KUKA KRL program: wkz3_ok.src, wkz3_ok.dat

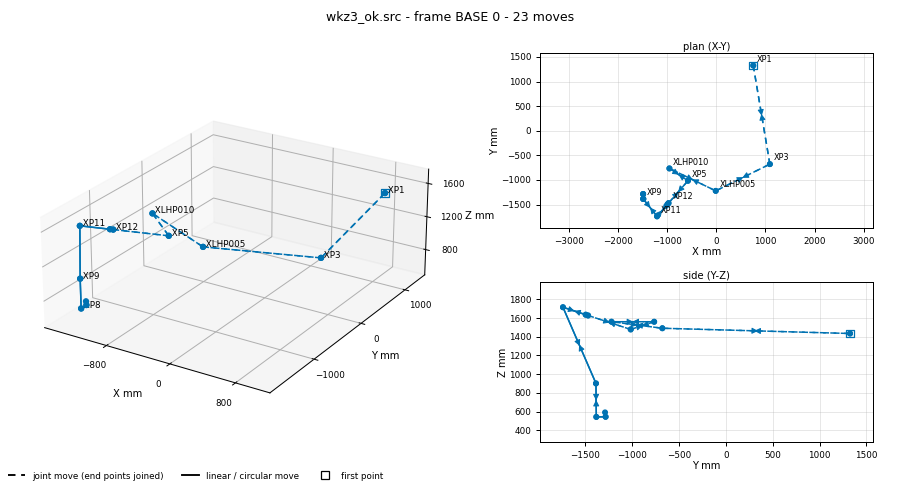
[picture p0: tool path of wkz3_ok.src in frame BASE 0, 23 of 23 moves have a stored position in this frame; points joined in program order, loops and branches not executed]
--- wkz3_ok.src ---
&ACCESS RVP
&REL 455
&COMMENT Check TCP C2
&PARAM DISKPATH = KRC:\R1\Program\TOOL CHANGE
&PARAM TEMPLATE = C:\KRC\Roboter\Template\vorgabe
&PARAM EDITMASK = *
DEF wkz3_ok( )
;FOLD INI
   ;FOLD BASISTECH INI
      GLOBAL INTERRUPT DECL 3 WHEN $STOPMESS==TRUE DO IR_STOPM ( )
      INTERRUPT ON 3
      BAS (#INITMOV,0 )
   ;ENDFOLD (BASISTECH INI)
   ;FOLD SPOTTECH INI
      USERSPOT(#INIT)
   ;ENDFOLD (SPOTTECH INI)
   ;FOLD GRIPPERTECH INI
      USER_GRP(0,DUMMY,DUMMY,GDEFAULT)
   ;ENDFOLD (GRIPPERTECH INI)
   ;FOLD USER INI
      ;Make your modifications here

   ;ENDFOLD (USER INI)
;ENDFOLD (INI)

; Estacao P13.060 - Robo R1
; Programa: Check TCP C2
; Caracterização dos meios de produção:
; 02/09/2014 09:15 Changes by KUKA Roboter do Brasil
;FOLD ; falta instalacao do check vertical;%{PE}%R 8.2.20,%MKUKATPBASIS,%CCOMMENT,%VNORMAL,%P 2:falta  instalacao  do  check  vertical
;ENDFOLD

chk_w3_wechs_ok ( )   ; CHECK FERRAMENTA: GUN C2

;FOLD PTP P1 Vel=100 % PDAT3 Tool[3]:GUN C2 Base[0];%{PE}%R 8.2.20,%MKUKATPBASIS,%CMOVE,%VPTP,%P 1:PTP, 2:P1, 3:, 5:100, 7:PDAT3
$BWDSTART=FALSE
PDAT_ACT=PPDAT3
FDAT_ACT=FP1
BAS(#PTP_PARAMS,100)
PTP XP1
;ENDFOLD
;FOLD PTP P3 Vel=100 % PDAT5 Tool[3]:GUN C2 Base[0];%{PE}%R 8.2.20,%MKUKATPBASIS,%CMOVE,%VPTP,%P 1:PTP, 2:P3, 3:, 5:100, 7:PDAT5
$BWDSTART=FALSE
PDAT_ACT=PPDAT5
FDAT_ACT=FP3
BAS(#PTP_PARAMS,100)
PTP XP3
;ENDFOLD
;FOLD PTP LHP005 CONT Vel=100 % PDAT1 Tool[3]:GUN C2 Base[0];%{PE}%R 8.2.20,%MKUKATPBASIS,%CMOVE,%VPTP,%P 1:PTP, 2:LHP005, 3:C_DIS, 5:100, 7:PDAT1
$BWDSTART=FALSE
PDAT_ACT=PPDAT1
FDAT_ACT=FLHP005
BAS(#PTP_PARAMS,100)
PTP XLHP005 C_DIS
;ENDFOLD
;FOLD PTP LHP010 CONT Vel=100 % PDAT2 Tool[3]:GUN C2 Base[0];%{PE}%R 8.2.20,%MKUKATPBASIS,%CMOVE,%VPTP,%P 1:PTP, 2:LHP010, 3:C_DIS, 5:100, 7:PDAT2
$BWDSTART=FALSE
PDAT_ACT=PPDAT2
FDAT_ACT=FLHP010
BAS(#PTP_PARAMS,100)
PTP XLHP010 C_DIS
;ENDFOLD
;FOLD PTP P5 CONT Vel=100 % PDAT20 Tool[3]:GUN C2 Base[0];%{PE}%R 8.2.20,%MKUKATPBASIS,%CMOVE,%VPTP,%P 1:PTP, 2:P5, 3:C_DIS, 5:100, 7:PDAT20
$BWDSTART=FALSE
PDAT_ACT=PPDAT20
FDAT_ACT=FP5
BAS(#PTP_PARAMS,100)
PTP XP5 C_DIS
;ENDFOLD
;FOLD PTP P12 CONT Vel=100 % PDAT25 Tool[3]:GUN C2 Base[0];%{PE}%R 8.2.20,%MKUKATPBASIS,%CMOVE,%VPTP,%P 1:PTP, 2:P12, 3:C_DIS, 5:100, 7:PDAT25
$BWDSTART=FALSE
PDAT_ACT=PPDAT25
FDAT_ACT=FP12
BAS(#PTP_PARAMS,100)
PTP XP12 C_DIS
;ENDFOLD
;FOLD LIN P13 CONT Vel=0.5 m/s CPDAT13 Tool[3]:GUN C2 Base[0];%{PE}%R 8.2.20,%MKUKATPBASIS,%CMOVE,%VLIN,%P 1:LIN, 2:P13, 3:C_DIS C_DIS, 5:0.5, 7:CPDAT13
$BWDSTART=FALSE
LDAT_ACT=LCPDAT13
FDAT_ACT=FP13
BAS(#CP_PARAMS,0.5)
LIN XP13 C_DIS C_DIS
;ENDFOLD
;FOLD LIN P11 CONT Vel=0.5 m/s CPDAT9 Tool[3]:GUN C2 Base[0];%{PE}%R 8.2.20,%MKUKATPBASIS,%CMOVE,%VLIN,%P 1:LIN, 2:P11, 3:C_DIS C_DIS, 5:0.5, 7:CPDAT9
$BWDSTART=FALSE
LDAT_ACT=LCPDAT9
FDAT_ACT=FP11
BAS(#CP_PARAMS,0.5)
LIN XP11 C_DIS C_DIS
;ENDFOLD
;FOLD LIN P9 CONT Vel=0.5 m/s CPDAT8 Tool[3]:GUN C2 Base[0];%{PE}%R 8.2.20,%MKUKATPBASIS,%CMOVE,%VLIN,%P 1:LIN, 2:P9, 3:C_DIS C_DIS, 5:0.5, 7:CPDAT8
$BWDSTART=FALSE
LDAT_ACT=LCPDAT8
FDAT_ACT=FP9
BAS(#CP_PARAMS,0.5)
LIN XP9 C_DIS C_DIS
;ENDFOLD
;FOLD LIN P8 CONT Vel=0.5 m/s CPDAT10 Tool[3]:GUN C2 Base[0];%{PE}%R 8.2.20,%MKUKATPBASIS,%CMOVE,%VLIN,%P 1:LIN, 2:P8, 3:C_DIS C_DIS, 5:0.5, 7:CPDAT10
$BWDSTART=FALSE
LDAT_ACT=LCPDAT10
FDAT_ACT=FP8
BAS(#CP_PARAMS,0.5)
LIN XP8 C_DIS C_DIS
;ENDFOLD
;FOLD LIN LHP015 Vel=0.5 m/s CPDAT3 Tool[3]:GUN C2 Base[0];%{PE}%R 8.2.20,%MKUKATPBASIS,%CMOVE,%VLIN,%P 1:LIN, 2:LHP015, 3:, 5:0.5, 7:CPDAT3
$BWDSTART=FALSE
LDAT_ACT=LCPDAT3
FDAT_ACT=FLHP015
BAS(#CP_PARAMS,0.5)
LIN XLHP015
;ENDFOLD

;FOLD ; posicao check tcp;%{PE}%R 4.1.16,%MKUKATPBASIS,%CCOMMENT,%VNORMAL,%P 2:posicao check tcp
;ENDFOLD
;FOLD LIN ChkTCPPos_Gun02 Vel=0.5 m/s CPDAT1 Tool[3]:GUN C2 Base[0];%{PE}%R 8.2.20,%MKUKATPBASIS,%CMOVE,%VLIN,%P 1:LIN, 2:ChkTCPPos_Gun02, 3:, 5:0.5, 7:CPDAT1
$BWDSTART=FALSE
LDAT_ACT=LCPDAT1
FDAT_ACT=FChkTCPPos_Gun02
BAS(#CP_PARAMS,0.5)
LIN XChkTCPPos_Gun02
;ENDFOLD
;FOLD WAIT Time= 5 sec;%{PE}%R 4.1.16,%MKUKATPBASIS,%CWAIT,%VWAIT,%P 2:5
WAIT SEC 5
;ENDFOLD

;FOLD LIN P7 CONT Vel=0.5 m/s CPDAT4 Tool[3]:GUN C2 Base[0];%{PE}%R 8.2.20,%MKUKATPBASIS,%CMOVE,%VLIN,%P 1:LIN, 2:P7, 3:C_DIS C_DIS, 5:0.5, 7:CPDAT4
$BWDSTART=FALSE
LDAT_ACT=LCPDAT4
FDAT_ACT=FP7
BAS(#CP_PARAMS,0.5)
LIN XP7 C_DIS C_DIS
;ENDFOLD
;FOLD LIN P14 CONT Vel=0.5 m/s CPDAT11 Tool[3]:GUN C2 Base[0];%{PE}%R 8.2.20,%MKUKATPBASIS,%CMOVE,%VLIN,%P 1:LIN, 2:P14, 3:C_DIS C_DIS, 5:0.5, 7:CPDAT11
$BWDSTART=FALSE
LDAT_ACT=LCPDAT11
FDAT_ACT=FP14
BAS(#CP_PARAMS,0.5)
LIN XP14 C_DIS C_DIS
;ENDFOLD
;FOLD LIN P15 CONT Vel=0.5 m/s CPDAT12 Tool[3]:GUN C2 Base[0];%{PE}%R 8.2.20,%MKUKATPBASIS,%CMOVE,%VLIN,%P 1:LIN, 2:P15, 3:C_DIS C_DIS, 5:0.5, 7:CPDAT12
$BWDSTART=FALSE
LDAT_ACT=LCPDAT12
FDAT_ACT=FP15
BAS(#CP_PARAMS,0.5)
LIN XP15 C_DIS C_DIS
;ENDFOLD
;FOLD LIN P16 CONT Vel=0.5 m/s CPDAT14 Tool[3]:GUN C2 Base[0];%{PE}%R 8.2.20,%MKUKATPBASIS,%CMOVE,%VLIN,%P 1:LIN, 2:P16, 3:C_DIS C_DIS, 5:0.5, 7:CPDAT14
$BWDSTART=FALSE
LDAT_ACT=LCPDAT14
FDAT_ACT=FP16
BAS(#CP_PARAMS,0.5)
LIN XP16 C_DIS C_DIS
;ENDFOLD
;FOLD LIN P17 CONT Vel=0.5 m/s CPDAT15 Tool[3]:GUN C2 Base[0];%{PE}%R 8.2.20,%MKUKATPBASIS,%CMOVE,%VLIN,%P 1:LIN, 2:P17, 3:C_DIS C_DIS, 5:0.5, 7:CPDAT15
$BWDSTART=FALSE
LDAT_ACT=LCPDAT15
FDAT_ACT=FP17
BAS(#CP_PARAMS,0.5)
LIN XP17 C_DIS C_DIS
;ENDFOLD
;FOLD LIN P18 CONT Vel=0.5 m/s CPDAT17 Tool[3]:GUN C2 Base[0];%{PE}%R 8.2.20,%MKUKATPBASIS,%CMOVE,%VLIN,%P 1:LIN, 2:P18, 3:C_DIS C_DIS, 5:0.5, 7:CPDAT17
$BWDSTART=FALSE
LDAT_ACT=LCPDAT17
FDAT_ACT=FP18
BAS(#CP_PARAMS,0.5)
LIN XP18 C_DIS C_DIS
;ENDFOLD
;FOLD PTP P19 CONT Vel=100 % PDAT27 Tool[3]:GUN C2 Base[0];%{PE}%R 8.2.20,%MKUKATPBASIS,%CMOVE,%VPTP,%P 1:PTP, 2:P19, 3:C_DIS, 5:100, 7:PDAT27
$BWDSTART=FALSE
PDAT_ACT=PPDAT27
FDAT_ACT=FP19
BAS(#PTP_PARAMS,100)
PTP XP19 C_DIS
;ENDFOLD
;FOLD PTP P20 CONT Vel=100 % PDAT28 Tool[3]:GUN C2 Base[0];%{PE}%R 8.2.20,%MKUKATPBASIS,%CMOVE,%VPTP,%P 1:PTP, 2:P20, 3:C_DIS, 5:100, 7:PDAT28
$BWDSTART=FALSE
PDAT_ACT=PPDAT28
FDAT_ACT=FP20
BAS(#PTP_PARAMS,100)
PTP XP20 C_DIS
;ENDFOLD
;FOLD PTP P21 CONT Vel=100 % PDAT29 Tool[3]:GUN C2 Base[0];%{PE}%R 8.2.20,%MKUKATPBASIS,%CMOVE,%VPTP,%P 1:PTP, 2:P21, 3:C_DIS, 5:100, 7:PDAT29
$BWDSTART=FALSE
PDAT_ACT=PPDAT29
FDAT_ACT=FP21
BAS(#PTP_PARAMS,100)
PTP XP21 C_DIS
;ENDFOLD
;FOLD PTP P22 CONT Vel=100 % PDAT30 Tool[3]:GUN C2 Base[0];%{PE}%R 8.2.20,%MKUKATPBASIS,%CMOVE,%VPTP,%P 1:PTP, 2:P22, 3:C_DIS, 5:100, 7:PDAT30
$BWDSTART=FALSE
PDAT_ACT=PPDAT30
FDAT_ACT=FP22
BAS(#PTP_PARAMS,100)
PTP XP22 C_DIS
;ENDFOLD
;FOLD PTP P23 CONT Vel=100 % PDAT31 Tool[3]:GUN C2 Base[0];%{PE}%R 8.2.20,%MKUKATPBASIS,%CMOVE,%VPTP,%P 1:PTP, 2:P23, 3:C_DIS, 5:100, 7:PDAT31
$BWDSTART=FALSE
PDAT_ACT=PPDAT31
FDAT_ACT=FP23
BAS(#PTP_PARAMS,100)
PTP XP23 C_DIS
;ENDFOLD
END

--- wkz3_ok.dat ---
&ACCESS RVP
&REL 455
&COMMENT Check TCP C2
&PARAM DISKPATH = KRC:\R1\Program\TOOL CHANGE
&PARAM TEMPLATE = C:\KRC\Roboter\Template\vorgabe
&PARAM EDITMASK = *
DEFDAT  wkz3_ok
;FOLD EXTERNAL DECLARATIONS;%{PE}%MKUKATPBASIS,%CEXT,%VCOMMON,%P
;FOLD GRIPPERTECH EXT
EXT  H50 (INT  :IN,INT  :IN,INT  :IN,GRP_TYP  :IN )
;ENDFOLD (GRIPPERTECH EXT)
;FOLD SPOTTECH EXT
EXT  USERSPOT (S_COMMAND  :IN,SPOT_TYPE  :IN )
;ENDFOLD (SPOTTECH EXT)
;FOLD BASISTECH EXT;%{PE}%MKUKATPBASIS,%CEXT,%VEXT,%P
EXT  BAS (BAS_COMMAND  :IN,REAL  :IN )
DECL INT SUCCESS
;ENDFOLD (BASISTECH EXT)
;FOLD USER EXT;%{E}%MKUKATPUSER,%CEXT,%VEXT,%P
;Make your modifications here

;ENDFOLD (USER EXT)
;ENDFOLD (EXTERNAL DECLARATIONS)

DECL PDAT PPDAT1={VEL 100.0,ACC 80.0,APO_DIST 10.0,APO_MODE #CDIS}
DECL E6POS XLHP010={X -951.651184,Y -765.088989,Z 1560.073,A -119.308197,B -41.8342018,C -84.1509628,S 18,T 2,E1 0.0,E2 0.0,E3 0.0,E4 0.0,E5 0.0,E6 0.0}
DECL FDAT FLHP010={TOOL_NO 3,BASE_NO 0,IPO_FRAME #BASE,TQ_STATE FALSE}
DECL PDAT PPDAT2={VEL 100.0,ACC 80.0,APO_DIST 10.0,APO_MODE #CDIS}
DECL E6POS XLHP015={X -1485.69995,Y -1283.427,Z 545.450623,A 90.8472366,B -0.687042773,C 0.235894397,S 18,T 10,E1 0.0,E2 0.0,E3 0.0,E4 0.0,E5 0.0,E6 0.0}
DECL FDAT FLHP015={TOOL_NO 3,BASE_NO 0,IPO_FRAME #BASE,TQ_STATE FALSE}
DECL E6POS XLHP020={X -1484.229,Y -1382.71899,Z 544.335388,A 90.8472672,B -0.689551473,C 0.235781297,S 18,T 10,E1 0.0,E2 0.0,E3 0.0,E4 0.0,E5 0.0,E6 0.0}
DECL FDAT FLHP020={TOOL_NO 3,BASE_NO 0,IPO_FRAME #BASE,TQ_STATE FALSE}
DECL E6POS XLHP025={X 1034.203,Y -165.537598,Z 959.119873,A -100.153702,B -15.1243601,C -86.5133896,S 18,T 2,E1 0.0,E2 0.0,E3 0.0,E4 0.0,E5 0.0,E6 0.0}
DECL FDAT FLHP025={TOOL_NO 3,BASE_NO 0,IPO_FRAME #BASE,TQ_STATE FALSE}
DECL PDAT PPDAT7={VEL 100.0,ACC 80.0,APO_DIST 10.0,APO_MODE #CDIS}
DECL E6POS XLHP030={X 1218.96802,Y 806.147278,Z 1597.64697,A 176.970596,B -2.82581401,C -90.4064636,S 18,T 3,E1 0.0,E2 0.0,E3 0.0,E4 0.0,E5 0.0,E6 0.0}
DECL FDAT FLHP030={TOOL_NO 3,BASE_NO 0,IPO_FRAME #BASE,TQ_STATE FALSE}
DECL PDAT PPDAT8={VEL 100.0,ACC 80.0,APO_DIST 10.0,APO_MODE #CDIS}
DECL PDAT PPDAT14={VEL 30.0,ACC 80.0,APO_DIST 10.0}
DECL PDAT PPDAT10={VEL 100.0,ACC 80.0,APO_DIST 10.0}
DECL PDAT PPDAT11={VEL 100.0,ACC 80.0,APO_DIST 10.0}
DECL E6POS XLHP005={X -10.4802904,Y -1220.74597,Z 1560.54199,A -68.6302338,B -41.8773613,C -84.0859604,S 18,T 2,E1 0.0,E2 0.0,E3 0.0,E4 0.0,E5 0.0,E6 0.0}
DECL FDAT FLHP005={TOOL_NO 3,BASE_NO 0,IPO_FRAME #BASE,TQ_STATE FALSE}
DECL E6POS XChkTCPPos_Gun02={X -1485.28503,Y -1289.51794,Z 592.772583,A 90.8463516,B -0.690602124,C 0.233830601,S 18,T 34,E1 0.0,E2 0.0,E3 0.0,E4 0.0,E5 0.0,E6 0.0}
DECL FDAT FChkTCPPos_Gun02={TOOL_NO 3,BASE_NO 0,IPO_FRAME #BASE,TQ_STATE FALSE}
DECL BASIS_SUGG_T LAST_BASIS={POINT1[] "P23                     ",POINT2[] "P23                     ",CP_PARAMS[] "CPDAT15                 ",PTP_PARAMS[] "PDAT31                  ",CONT[] "C_DIS                   ",CP_VEL[] "0.5                     ",PTP_VEL[] "100                     ",SYNC_PARAMS[] "SYNCDAT                 ",SPL_NAME[] "S0                      "}
DECL E6POS XP1={X 752.183289,Y 1325.57202,Z 1434.74805,A 80.377739,B -52.962841,C -87.0940628,S 18,T 3,E1 0.0,E2 0.0,E3 0.0,E4 0.0,E5 0.0,E6 0.0}
DECL FDAT FP1={TOOL_NO 3,BASE_NO 0,IPO_FRAME #BASE,POINT2[] " ",TQ_STATE FALSE}
DECL PDAT PPDAT3={VEL 100.0,ACC 100.0,APO_DIST 100.0,APO_MODE #CDIS,GEAR_JERK 50.0}
DECL E6POS XP2={X 752.183411,Y 1325.57202,Z 1434.74805,A 80.3777237,B -52.9628296,C -87.0940475,S 18,T 3,E1 0.0,E2 0.0,E3 0.0,E4 0.0,E5 0.0,E6 0.0}
DECL FDAT FP2={TOOL_NO 3,BASE_NO 0,IPO_FRAME #BASE,POINT2[] " ",TQ_STATE FALSE}
DECL PDAT PPDAT4={VEL 100.0,ACC 100.0,APO_DIST 100.0,APO_MODE #CDIS,GEAR_JERK 50.0}
DECL E6POS XP3={X 1089.15002,Y -677.833313,Z 1490.74402,A -17.2367191,B -46.5962105,C -77.8356628,S 18,T 3,E1 0.0,E2 0.0,E3 0.0,E4 0.0,E5 0.0,E6 0.0}
DECL FDAT FP3={TOOL_NO 3,BASE_NO 0,IPO_FRAME #BASE,POINT2[] " ",TQ_STATE FALSE}
DECL PDAT PPDAT5={VEL 100.0,ACC 100.0,APO_DIST 100.0,APO_MODE #CDIS,GEAR_JERK 50.0}
DECL E6POS XP4={X 846.179504,Y 853.370178,Z 1095.526,A -43.7265511,B -17.3734303,C -31.7438393,S 18,T 3,E1 0.0,E2 0.0,E3 0.0,E4 0.0,E5 0.0,E6 0.0}
DECL FDAT FP4={TOOL_NO 3,BASE_NO 0,IPO_FRAME #BASE,POINT2[] " ",TQ_STATE FALSE}
DECL PDAT PPDAT6={VEL 100.0,ACC 100.0,APO_DIST 100.0,APO_MODE #CDIS,GEAR_JERK 50.0}
DECL LDAT LCPDAT1={VEL 2.0,ACC 100.0,APO_DIST 100.0,APO_FAC 50.0,AXIS_VEL 100.0,AXIS_ACC 100.0,ORI_TYP #VAR,CIRC_TYP #BASE,JERK_FAC 50.0,GEAR_JERK 50.0,EXAX_IGN 0}
DECL LDAT LCPDAT2={VEL 2.0,ACC 100.0,APO_DIST 100.0,APO_FAC 50.0,AXIS_VEL 100.0,AXIS_ACC 100.0,ORI_TYP #VAR,CIRC_TYP #BASE,JERK_FAC 50.0,GEAR_JERK 50.0,EXAX_IGN 0}
DECL E6POS XP5={X -575.287415,Y -1015.63702,Z 1478.19995,A 147.233505,B -13.7448502,C -19.7403297,S 18,T 2,E1 0.0,E2 0.0,E3 0.0,E4 0.0,E5 0.0,E6 0.0}
DECL FDAT FP5={TOOL_NO 3,BASE_NO 0,IPO_FRAME #BASE,POINT2[] " ",TQ_STATE FALSE}
DECL PDAT PPDAT9={VEL 100.0,ACC 80.0,APO_DIST 10.0,APO_MODE #CDIS,GEAR_JERK 50.0}
DECL LDAT LCPDAT3={VEL 2.0,ACC 100.0,APO_DIST 100.0,APO_FAC 50.0,AXIS_VEL 100.0,AXIS_ACC 100.0,ORI_TYP #VAR,CIRC_TYP #BASE,JERK_FAC 50.0,GEAR_JERK 50.0,EXAX_IGN 0}
DECL E6POS XP6={X -1484.27502,Y -1382.76001,Z 544.360779,A 90.8475113,B -0.68821919,C 0.236860305,S 18,T 10,E1 0.0,E2 0.0,E3 0.0,E4 0.0,E5 0.0,E6 0.0}
DECL FDAT FP6={TOOL_NO 3,BASE_NO 0,IPO_FRAME #BASE,POINT2[] " ",TQ_STATE FALSE}
DECL PDAT PPDAT12={VEL 100.0,ACC 80.0,APO_DIST 10.0,APO_MODE #CDIS,GEAR_JERK 50.0}
DECL PDAT PPDAT13={VEL 100.0,ACC 80.0,APO_DIST 10.0,APO_MODE #CDIS,GEAR_JERK 50.0}
DECL E6POS XP7={X -1485.68396,Y -1283.41394,Z 545.442078,A 90.8471222,B -0.687304497,C 0.2354801,S 18,T 10,E1 0.0,E2 0.0,E3 0.0,E4 0.0,E5 0.0,E6 0.0}
DECL FDAT FP7={TOOL_NO 3,BASE_NO 0,IPO_FRAME #BASE,POINT2[] " ",TQ_STATE FALSE}
DECL LDAT LCPDAT4={VEL 2.0,ACC 100.0,APO_DIST 100.0,APO_FAC 50.0,AXIS_VEL 100.0,AXIS_ACC 100.0,ORI_TYP #VAR,CIRC_TYP #BASE,JERK_FAC 50.0,GEAR_JERK 50.0,EXAX_IGN 0}
DECL E6POS XP8={X -1484.24304,Y -1382.73206,Z 544.342285,A 90.8473663,B -0.689165771,C 0.236065507,S 18,T 10,E1 0.0,E2 0.0,E3 0.0,E4 0.0,E5 0.0,E6 0.0}
DECL FDAT FP8={TOOL_NO 3,BASE_NO 0,IPO_FRAME #BASE,POINT2[] " ",TQ_STATE FALSE}
DECL PDAT PPDAT15={VEL 100.0,ACC 80.0,APO_DIST 10.0,APO_MODE #CDIS,GEAR_JERK 50.0}
DECL E6POS XP9={X -1481.99695,Y -1386.32898,Z 901.916687,A 90.8413467,B -0.701726079,C 0.231831402,S 18,T 10,E1 0.0,E2 0.0,E3 0.0,E4 0.0,E5 0.0,E6 0.0}
DECL FDAT FP9={TOOL_NO 3,BASE_NO 0,IPO_FRAME #BASE,POINT2[] " ",TQ_STATE FALSE}
DECL PDAT PPDAT16={VEL 100.0,ACC 80.0,APO_DIST 10.0,APO_MODE #CDIS,GEAR_JERK 50.0}
DECL E6POS XP10={X -1481.98499,Y -1386.31799,Z 901.909607,A 90.8412399,B -0.702053726,C 0.231592193,S 18,T 10,E1 0.0,E2 0.0,E3 0.0,E4 0.0,E5 0.0,E6 0.0}
DECL FDAT FP10={TOOL_NO 3,BASE_NO 0,IPO_FRAME #BASE,POINT2[] " ",TQ_STATE FALSE}
DECL PDAT PPDAT17={VEL 100.0,ACC 80.0,APO_DIST 10.0,APO_MODE #CDIS,GEAR_JERK 50.0}
DECL E6POS XP11={X -1202.98206,Y -1738.68005,Z 1715.09094,A 123.543999,B 20.3694496,C 22.7444096,S 18,T 10,E1 0.0,E2 0.0,E3 0.0,E4 0.0,E5 0.0,E6 0.0}
DECL FDAT FP11={TOOL_NO 3,BASE_NO 0,IPO_FRAME #BASE,POINT2[] " ",TQ_STATE FALSE}
DECL PDAT PPDAT18={VEL 100.0,ACC 80.0,APO_DIST 10.0,APO_MODE #CDIS,GEAR_JERK 50.0}
DECL LDAT LCPDAT5={VEL 2.0,ACC 100.0,APO_DIST 100.0,APO_FAC 50.0,AXIS_VEL 100.0,AXIS_ACC 100.0,ORI_TYP #VAR,CIRC_TYP #BASE,JERK_FAC 50.0,GEAR_JERK 50.0,EXAX_IGN 0}
DECL LDAT LCPDAT6={VEL 2.0,ACC 100.0,APO_DIST 100.0,APO_FAC 50.0,AXIS_VEL 100.0,AXIS_ACC 100.0,ORI_TYP #VAR,CIRC_TYP #BASE,JERK_FAC 50.0,GEAR_JERK 50.0,EXAX_IGN 0}
DECL E6POS XP12={X -969.846191,Y -1470.16003,Z 1626.94702,A 132.607101,B 7.80172586,C 8.64788532,S 18,T 34,E1 0.0,E2 0.0,E3 0.0,E4 0.0,E5 0.0,E6 0.0}
DECL FDAT FP12={TOOL_NO 3,BASE_NO 0,IPO_FRAME #BASE,POINT2[] " ",TQ_STATE FALSE}
DECL PDAT PPDAT19={VEL 100.0,ACC 80.0,APO_DIST 10.0,APO_MODE #CDIS,GEAR_JERK 50.0}
DECL PDAT PPDAT20={VEL 100.0,ACC 80.0,APO_DIST 10.0,APO_MODE #CDIS,GEAR_JERK 50.0}
DECL PDAT PPDAT21={VEL 100.0,ACC 80.0,APO_DIST 10.0,APO_MODE #CDIS,GEAR_JERK 50.0}
DECL LDAT LCPDAT7={VEL 2.0,ACC 100.0,APO_DIST 100.0,APO_FAC 50.0,AXIS_VEL 100.0,AXIS_ACC 100.0,ORI_TYP #VAR,CIRC_TYP #BASE,JERK_FAC 50.0,GEAR_JERK 50.0,EXAX_IGN 0}
DECL E6POS XP13={X -992.084717,Y -1496.15601,Z 1635.505,A 131.764496,B 9.02914524,C 10.0937901,S 18,T 34,E1 0.0,E2 0.0,E3 0.0,E4 0.0,E5 0.0,E6 0.0}
DECL FDAT FP13={TOOL_NO 3,BASE_NO 0,IPO_FRAME #BASE,POINT2[] " ",TQ_STATE FALSE}
DECL PDAT PPDAT22={VEL 100.0,ACC 80.0,APO_DIST 10.0,APO_MODE #CDIS,GEAR_JERK 50.0}
DECL PDAT PPDAT23={VEL 100.0,ACC 80.0,APO_DIST 10.0,APO_MODE #CDIS,GEAR_JERK 50.0}
DECL LDAT LCPDAT8={VEL 2.0,ACC 100.0,APO_DIST 100.0,APO_FAC 50.0,AXIS_VEL 100.0,AXIS_ACC 100.0,ORI_TYP #VAR,CIRC_TYP #BASE,JERK_FAC 50.0,GEAR_JERK 50.0,EXAX_IGN 0}
DECL LDAT LCPDAT9={VEL 2.0,ACC 100.0,APO_DIST 100.0,APO_FAC 50.0,AXIS_VEL 100.0,AXIS_ACC 100.0,ORI_TYP #VAR,CIRC_TYP #BASE,JERK_FAC 50.0,GEAR_JERK 50.0,EXAX_IGN 0}
DECL LDAT LCPDAT10={VEL 2.0,ACC 100.0,APO_DIST 100.0,APO_FAC 50.0,AXIS_VEL 100.0,AXIS_ACC 100.0,ORI_TYP #VAR,CIRC_TYP #BASE,JERK_FAC 50.0,GEAR_JERK 50.0,EXAX_IGN 0}
DECL E6POS XP14={X -1484.25696,Y -1382.78601,Z 544.375488,A 90.8466415,B -0.683399618,C 0.237654194,S 18,T 10,E1 0.0,E2 0.0,E3 0.0,E4 0.0,E5 0.0,E6 0.0}
DECL FDAT FP14={TOOL_NO 3,BASE_NO 0,IPO_FRAME #BASE,POINT2[] " ",TQ_STATE FALSE}
DECL LDAT LCPDAT11={VEL 2.0,ACC 100.0,APO_DIST 100.0,APO_FAC 50.0,AXIS_VEL 100.0,AXIS_ACC 100.0,ORI_TYP #VAR,CIRC_TYP #BASE,JERK_FAC 50.0,GEAR_JERK 50.0,EXAX_IGN 0}
DECL E6POS XP15={X -1481.979,Y -1386.33997,Z 901.907776,A 90.8411102,B -0.700398624,C 0.231303602,S 18,T 10,E1 0.0,E2 0.0,E3 0.0,E4 0.0,E5 0.0,E6 0.0}
DECL FDAT FP15={TOOL_NO 3,BASE_NO 0,IPO_FRAME #BASE,POINT2[] " ",TQ_STATE FALSE}
DECL LDAT LCPDAT12={VEL 2.0,ACC 100.0,APO_DIST 100.0,APO_FAC 50.0,AXIS_VEL 100.0,AXIS_ACC 100.0,ORI_TYP #VAR,CIRC_TYP #BASE,JERK_FAC 50.0,GEAR_JERK 50.0,EXAX_IGN 0}
DECL E6POS XP16={X -1202.97998,Y -1738.67004,Z 1715.08801,A 123.5439,B 20.3694191,C 22.7444897,S 18,T 10,E1 0.0,E2 0.0,E3 0.0,E4 0.0,E5 0.0,E6 0.0}
DECL FDAT FP16={TOOL_NO 3,BASE_NO 0,IPO_FRAME #BASE,POINT2[] " ",TQ_STATE FALSE}
DECL PDAT PPDAT24={VEL 100.0,ACC 80.0,APO_DIST 10.0,APO_MODE #CDIS,GEAR_JERK 50.0}
DECL LDAT LCPDAT13={VEL 2.0,ACC 100.0,APO_DIST 100.0,APO_FAC 50.0,AXIS_VEL 100.0,AXIS_ACC 100.0,ORI_TYP #VAR,CIRC_TYP #BASE,JERK_FAC 50.0,GEAR_JERK 50.0,EXAX_IGN 0}
DECL LDAT LCPDAT14={VEL 2.0,ACC 100.0,APO_DIST 100.0,APO_FAC 50.0,AXIS_VEL 100.0,AXIS_ACC 100.0,ORI_TYP #VAR,CIRC_TYP #BASE,JERK_FAC 50.0,GEAR_JERK 50.0,EXAX_IGN 0}
DECL E6POS XP17={X -992.090881,Y -1496.14502,Z 1635.49805,A 131.764099,B 9.02908993,C 10.0937996,S 18,T 10,E1 0.0,E2 0.0,E3 0.0,E4 0.0,E5 0.0,E6 0.0}
DECL FDAT FP17={TOOL_NO 3,BASE_NO 0,IPO_FRAME #BASE,POINT2[] " ",TQ_STATE FALSE}
DECL LDAT LCPDAT15={VEL 2.0,ACC 100.0,APO_DIST 100.0,APO_FAC 50.0,AXIS_VEL 100.0,AXIS_ACC 100.0,ORI_TYP #VAR,CIRC_TYP #BASE,JERK_FAC 50.0,GEAR_JERK 50.0,EXAX_IGN 0}
DECL LDAT LCPDAT16={VEL 2.0,ACC 100.0,APO_DIST 100.0,APO_FAC 50.0,AXIS_VEL 100.0,AXIS_ACC 100.0,ORI_TYP #VAR,CIRC_TYP #BASE,JERK_FAC 50.0,GEAR_JERK 50.0,EXAX_IGN 0}
DECL PDAT PPDAT25={VEL 100.0,ACC 80.0,APO_DIST 10.0,APO_MODE #CDIS,GEAR_JERK 50.0}
DECL E6POS XP18={X -969.570984,Y -1470.151,Z 1626.94604,A 132.604507,B 7.79787683,C 8.63807774,S 18,T 34,E1 0.0,E2 0.0,E3 0.0,E4 0.0,E5 0.0,E6 0.0}
DECL FDAT FP18={TOOL_NO 3,BASE_NO 0,IPO_FRAME #BASE,POINT2[] " ",TQ_STATE FALSE}
DECL PDAT PPDAT26={VEL 100.0,ACC 80.0,APO_DIST 10.0,APO_MODE #CDIS,GEAR_JERK 50.0}
DECL E6POS XP19={X -575.289978,Y -1015.62701,Z 1478.19702,A 147.233398,B -13.74506,C -19.7406406,S 18,T 2,E1 0.0,E2 0.0,E3 0.0,E4 0.0,E5 0.0,E6 0.0}
DECL FDAT FP19={TOOL_NO 3,BASE_NO 0,IPO_FRAME #BASE,POINT2[] " ",TQ_STATE FALSE}
DECL PDAT PPDAT27={VEL 100.0,ACC 80.0,APO_DIST 10.0,APO_MODE #CDIS,GEAR_JERK 50.0}
DECL E6POS XP20={X -951.635925,Y -765.080627,Z 1560.05896,A -119.315102,B -41.8366089,C -84.1466904,S 18,T 2,E1 0.0,E2 0.0,E3 0.0,E4 0.0,E5 0.0,E6 0.0}
DECL FDAT FP20={TOOL_NO 3,BASE_NO 0,IPO_FRAME #BASE,POINT2[] " ",TQ_STATE FALSE}
DECL PDAT PPDAT28={VEL 100.0,ACC 80.0,APO_DIST 10.0,APO_MODE #CDIS,GEAR_JERK 50.0}
DECL E6POS XP21={X -10.4820404,Y -1220.74402,Z 1560.54102,A -68.630188,B -41.8770103,C -84.0861435,S 18,T 2,E1 0.0,E2 0.0,E3 0.0,E4 0.0,E5 0.0,E6 0.0}
DECL FDAT FP21={TOOL_NO 3,BASE_NO 0,IPO_FRAME #BASE,POINT2[] " ",TQ_STATE FALSE}
DECL PDAT PPDAT29={VEL 100.0,ACC 80.0,APO_DIST 10.0,APO_MODE #CDIS,GEAR_JERK 50.0}
DECL E6POS XP22={X 1089.13599,Y -677.836914,Z 1490.745,A -17.2370491,B -46.595871,C -77.8357773,S 18,T 3,E1 0.0,E2 0.0,E3 0.0,E4 0.0,E5 0.0,E6 0.0}
DECL FDAT FP22={TOOL_NO 3,BASE_NO 0,IPO_FRAME #BASE,POINT2[] " ",TQ_STATE FALSE}
DECL PDAT PPDAT30={VEL 100.0,ACC 80.0,APO_DIST 10.0,APO_MODE #CDIS,GEAR_JERK 50.0}
DECL E6POS XP23={X 752.1828,Y 1325.53601,Z 1434.72498,A 80.3768997,B -52.960331,C -87.0938797,S 18,T 3,E1 0.0,E2 0.0,E3 0.0,E4 0.0,E5 0.0,E6 0.0}
DECL FDAT FP23={TOOL_NO 3,BASE_NO 0,IPO_FRAME #BASE,POINT2[] " ",TQ_STATE FALSE}
DECL PDAT PPDAT31={VEL 100.0,ACC 80.0,APO_DIST 10.0,APO_MODE #CDIS,GEAR_JERK 50.0}
DECL LDAT LCPDAT17={VEL 2.0,ACC 100.0,APO_DIST 100.0,APO_FAC 50.0,AXIS_VEL 100.0,AXIS_ACC 100.0,ORI_TYP #VAR,CIRC_TYP #BASE,JERK_FAC 50.0,GEAR_JERK 50.0,EXAX_IGN 0}
ENDDAT
